// Mitsubishi GX Works2 project: 블록기동1   PLC: Q02/Q02H

PROGRAM MAIN
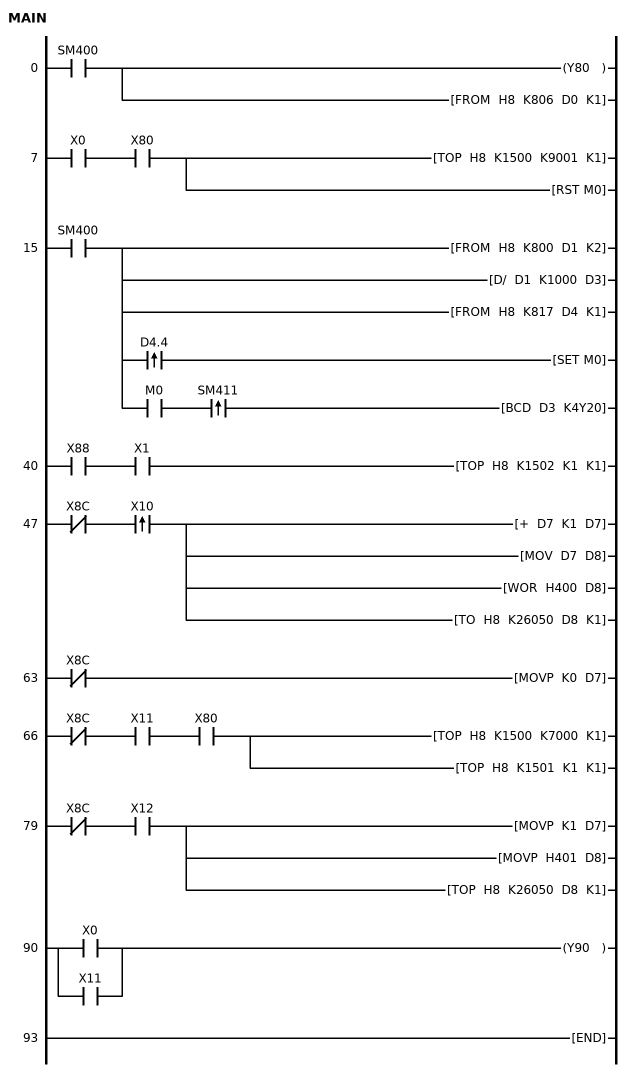
0     LD      SM400
      OUT     Y80
      FROM    H8 K806 D0 K1
7     LD      X0
      AND     X80
      TOP     H8 K1500 K9001 K1
      RST     M0
15    LD      SM400
      FROM    H8 K800 D1 K2
      D/      D1 K1000 D3
      FROM    H8 K817 D4 K1
      MPS
      ANDP    D4.4
      SET     M0
      MPP
      AND     M0
      ANDP    SM411
      BCD     D3 K4Y20
40    LD      X88
      AND     X1
      TOP     H8 K1502 K1 K1
47    LDI     X8C
      ANDP    X10
      +       D7 K1 D7
      MOV     D7 D8
      WOR     H400 D8
      TO      H8 K26050 D8 K1
63    LDI     X8C
      MOVP    K0 D7
66    LDI     X8C
      AND     X11
      AND     X80
      TOP     H8 K1500 K7000 K1
      TOP     H8 K1501 K1 K1
79    LDI     X8C
      AND     X12
      MOVP    K1 D7
      MOVP    H401 D8
      TOP     H8 K26050 D8 K1
90    LD      X0
      OR      X11
      OUT     Y90
93    END
END_PROGRAM
